(* IEC 61131-3 sources: AxTestProject/LStandardLibrary/Motion/Axis, 4 files *)

(* ---- eAxis.st ---- *)
NAMESPACE stdLib.Motion
    TYPE
        enStatus : STRUCT
            done : BOOL;
            busy : BOOL;
            error : BOOL;
            status : INT;
        END_STRUCT;
    END_TYPE
END_NAMESPACE

(* ---- tAxisStatus.st ---- *)
NAMESPACE stdLib.Motion
    TYPE
        tAxisStatus : STRUCT
            actPosition : DINT;
            isRunning : BOOL;
            hasFault : BOOL;
        END_STRUCT;
    END_TYPE

    //TYPE
    //    arrayOfStruct : ARRAY[0..1] of tAxisStatus := ;
    //END_TYPE

END_NAMESPACE

(* ---- AxisTest_MoveVelocity.st ---- *)
//{Test(fault:=false, resBusy:=true, resErr:=false)}
//{Test(fault:=true, resBusy:=false, resErr:=true)}
{Test}
FUNCTION moveVelocityRunOk
    VAR_INPUT
       fault : BOOL;
       resBusy : BOOL;
       resErr : BOOL;
    END_VAR
    VAR_TEMP
        res2 : BOOL;
        axis : stdLib.Motion.Axis;
        status : stdLib.Motion.enStatus;
        //boFault : BOOL;
    END_VAR

    //boFault := fault <> 0;

    axis.faultActive := false;
    res2 := axis.MoveVelocity();
    status := axis.GetStatus();

    Assert_Equal_BOOL(expected:=true, actual:=status.busy);
    Assert_Equal_BOOL(expected:=false, actual:=status.error);
    Assert_Equal_BOOL(expected:=false, actual:=status.done);

END_FUNCTION

{Test}
FUNCTION moveVelocityRunFalse
    VAR_TEMP
        res : BOOL;
        axis : stdLib.Motion.Axis;
        status : stdLib.Motion.enStatus;
    END_VAR

    axis.faultActive := true;
    res := axis.MoveVelocity();
    status := axis.GetStatus();

    Assert_Equal_BOOL(expected:=false, actual:=status.busy);
    Assert_Equal_BOOL(expected:=true, actual:=status.error);
    Assert_Equal_BOOL(expected:=false, actual:=status.done);

END_FUNCTION

(* ---- Axis.st ---- *)
NAMESPACE stdLib.Motion
    CLASS Axis

        VAR PUBLIC
            mParameter : stdLib.Motion.tAxisParameter;
            m1 : stdLib.Motion.tAxisParameter;
            mStatus : stdLib.Motion.tAxisStatus;
            run : BOOL;
            faultActive : BOOL;
        END_VAR

        VAR PRIVATE
            mPosition : DINT;
            mAcceleration : LREAL;
            mDeceleration : LREAL;
            mPlcOpenStatus : stdLib.Motion.enStatus;
        END_VAR

        METHOD PUBLIC Main
            ;
        END_METHOD

        METHOD PUBLIC  GetStatus : stdLib.Motion.enStatus
            GetStatus := mPlcOpenStatus;
        END_METHOD

        METHOD PUBLIC  GetInfo : stdLib.Motion.tAxisStatus
            GetInfo := mStatus;
        END_METHOD

        METHOD PUBLIC GetPos : DINT
            GetPos := mPosition;
        END_METHOD

        //--------------------------------------
        // Homing
        //--------------------------------------
        METHOD PUBLIC Homing : stdLib.Motion.enStatus
            VAR_INPUT
                //velocity : LREAL;
                //acceleration : LREAL;
                //deceleration : LREAL;
                //mode : INT;
            END_VAR
            VAR_TEMP
                tempStatus : stdLib.Motion.enStatus;
            END_VAR
                Homing := tempStatus;
        END_METHOD

        METHOD PRIVATE mHoming
            ;
        END_METHOD

        //---------------------------------------------------
        // Reset
        //---------------------------------------------------
        METHOD Reset : BOOL
            VAR_INPUT
            END_VAR
            VAR_TEMP
            END_VAR

            Reset := true;
                ;
        END_METHOD

        //---------------------------------------------------
        // Halt
        //---------------------------------------------------
        METHOD Halt : BOOL
            VAR_INPUT
            END_VAR
            VAR_TEMP
            END_VAR

            Halt := true;
                ;
        END_METHOD

        //---------------------------------------------------
        // MoveVelocity
        //---------------------------------------------------
        METHOD PUBLIC MoveVelocity : BOOL
            VAR_INPUT
                velocity : LREAL;
                acceleration : LREAL;
                deceleration : LREAL;
            END_VAR

            if (not(faultActive)) then
                mPlcOpenstatus.busy := true;
                MoveVelocity := true;
            ELSE
                mPlcOpenstatus.error := true;
                mPlcOpenstatus.busy := false;
                MoveVelocity := false;
            END_IF;

        END_METHOD

        //---------------------------------------------------
        // MoveAbsolute
        //---------------------------------------------------
        METHOD PUBLIC MoveAbsolute : BOOL
            VAR_INPUT
                velocity : LREAL;
                position : DINT;
                acceleration : LREAL;
                deceleration : LREAL;
            END_VAR
            MoveAbsolute := true;
        END_METHOD

        METHOD PUBLIC MoveAbsolute3 : BOOL
            VAR_INPUT
                velocity : LREAL;
                position : DINT;
                acceleration : LREAL;
                deceleration : LREAL;
            END_VAR
            MoveAbsolute3 := true;
        END_METHOD

        //---------------------------------------------------
        // MoveRelative
        //---------------------------------------------------
        METHOD PUBLIC MoveRelative : BOOL
            VAR_INPUT
                velocity : LREAL;
                position : DINT;
                acceleration : LREAL;
                deceleration : LREAL;
            END_VAR
            MoveRelative := true;
        END_METHOD

        //---------------------------------------------------
        // SetAcceleration
        //---------------------------------------------------
        METHOD PUBLIC SetAcceleration
            VAR_INPUT
                accelleration : LREAL;
            END_VAR
            mAcceleration := accelleration;
        END_METHOD

        //---------------------------------------------------
        // SetDeceleration
        //---------------------------------------------------
        METHOD PUBLIC SetDeceleration
            VAR_INPUT
                deceleration : LREAL;
            END_VAR
            mDeceleration := deceleration;
        END_METHOD

        METHOD init
            VAR_INPUT
                parameter : stdLib.Motion.tAxisParameter;
            END_VAR
            ;
            parameter.velocity := 0.0;
            parameter.position := DINT#0;
        END_METHOD

    END_CLASS
END_NAMESPACE
